Staubli VAL3: WeldTraj.pgx

program WeldTraj(bool& x_bRes)
  local num l_nId
  local num l_nBuffID
  local num l_nSize
  local num l_nNum
  local trsf l_trTrsf
begin
  //计算回退点
  l_nId=getMoveId()

  call Algorith:GetWeldReturn(TxtFile:pCut,TxtFile:pMoveC,TxtFile:bMoveC,l_nId,l_nBuffID,TxtFile:trIODelay.z,x_bRes)
  if !x_bRes or l_nBuffID<1  or l_nBuffID>(l_nId+0.0001)
   // popUpMsg(toString(".3",l_nBuffID))
    x_bRes=false
    return
  endIf

  if roundDown(l_nBuffID)==roundUp(l_nBuffID)
    l_nBuffID=l_nBuffID+0.0001
  endIf


  //圆弧

  if TxtFile:bMoveC[roundDown(l_nBuffID)]

    l_trTrsf=interpolateC(TxtFile:pCut[roundDown((l_nBuffID)-1)].trsf,TxtFile:pMoveC[roundDown(l_nBuffID)].trsf,TxtFile:pCut[roundDown(l_nBuffID)].trsf,l_nBuffID-roundDown(l_nBuffID))
  else

    l_trTrsf=interpolateL(TxtFile:pCut[roundDown((l_nBuffID)-1)].trsf,TxtFile:pCut[roundDown(l_nBuffID)].trsf,l_nBuffID-roundDown(l_nBuffID))
  endIf



  l_nSize=roundUp(l_nId)-roundDown(l_nBuffID)


  resize(TxtFile:jAppro,1,l_nSize)
  resize(TxtFile:pAppro,1,l_nSize)
  resize(TxtFile:trAppro,1,l_nSize)
  resize(TxtFile:bAppro,1,l_nSize)

  for l_nNum=0 to size(TxtFile:pAppro)-2
    TxtFile:bAppro[l_nNum]=true
    TxtFile:pAppro[l_nNum].trsf=TxtFile:pCut[roundDown(l_nId)-1-l_nNum].trsf
    TxtFile:trAppro[l_nNum]=TxtFile:trCut[roundDown(l_nId)-l_nNum-1]
  endFor

  TxtFile:pAppro[size(TxtFile:pAppro)-1].trsf=l_trTrsf
  TxtFile:bAppro[size(TxtFile:pAppro)-1]=true
  TxtFile:trAppro[size(TxtFile:pAppro)-1]=TxtFile:trAppro[0]

  for l_nNum=0 to roundDown(l_nBuffID)-2
    delete(TxtFile:pCut[0])
    delete(TxtFile:pMoveC[0])
    delete(TxtFile:trCut[0])
    delete(TxtFile:bMoveC[0])
  endFor
  TxtFile:pCut[0].trsf=l_trTrsf
  TxtFile:bMoveC[0]=false

  TxtFile:trPointCount.x=size(TxtFile:jAppro)
  TxtFile:trPointCount.y=size(TxtFile:pCut)

  x_bRes=true



end
